{attribute 'GeneratedUsingTerminal: BK1150-0000-0017'}
{attribute addProperty BoxType "BK1150-0000-0017"}
{attribute addProperty Id "Term_384_KL1002KL1002_BB38DA8F0"}
{attribute addProperty CRC "1067260198"}
{attribute addProperty Size "0"}
TYPE A_0011_BK1150_0000_0017_3F9D1926 EXTENDS BK1150_A2FCADE7 :
STRUCT
	{attribute addProperty Name "Term_384_KL1002"}
	Term_384_KL1002 : KL1002_BB38DA8F;
END_STRUCT
END_TYPE

(* stored: Version 1.2.0.0, ProductVersion 3.1.4024.9
   DUT A_0011_BK1150_0000_0017_3F9D1926: Id {8a665119-4a9c-41ec-85d7-ccfca4794ca6} *)
